PROGRAM MoveExtPos
VAR
	armState	:UINT:=0;
	chabustate	:UINT:=0;
	
	LeftArm_Right_ExtPosGen_Enable						:MC_ExtSetPointGenEnable;
	LeftArm_Right_ExtPosGen_Disable                     :MC_ExtSetPointGenDisable;
	LeftArm_Left_ExtPosGen_Enable                       :MC_ExtSetPointGenEnable;
	LeftArm_Left_ExtPosGen_Disable	                    :MC_ExtSetPointGenDisable;
	LeftArm_Wrist_ExtPosGen_Enable                      :MC_ExtSetPointGenEnable;
	LeftArm_Wrist_ExtPosGen_Disable	                    :MC_ExtSetPointGenDisable;
	
	RightArm_Right_ExtPosGen_Enable						:MC_ExtSetPointGenEnable;
	RightArm_Right_ExtPosGen_Disable                     :MC_ExtSetPointGenDisable;
	RightArm_Left_ExtPosGen_Enable                       :MC_ExtSetPointGenEnable;
	RightArm_Left_ExtPosGen_Disable	                    :MC_ExtSetPointGenDisable;
	RightArm_Wrist_ExtPosGen_Enable                      :MC_ExtSetPointGenEnable;
	RightArm_Wrist_ExtPosGen_Disable	                    :MC_ExtSetPointGenDisable;
	
	currentPosition_LeftArm				:Points;
	currentPosition_RightArm				:Points;

	//leftpoints						:ARRAY[0..5,0..1] OF LREAL:=[[-80,390],[390,880],[-80,390],[-80,880],[-80,390],[-400,830]];
	//rightpoints						:ARRAY[0..5,0..1] OF LREAL:=[[-80,390],[390,880],[-80,390],[-80,880],[-80,390],[-400,830]];	
	LeftArmWristTargetPos				:REAL;
	RightArmWristTargetPos				:REAL;	
	
	t			:LREAL:=0;
	delta_t		:LREAL:=0.0005;
	lx:LREAL;
	ly:LREAL;
	rx:LREAL;
	ry:LREAL;
	
	LeftArmAngle			:Angles;
	RightArmAngle			:Angles;


	
	

END_VAR

axis_LeftArm_Left();
axis_LeftArm_Right();
axis_LeftArm_Wrist();
axis_RightArm_Left();
axis_RightArm_Right();
axis_RightArm_Wrist();
ACT_ExtGen();


// 外部位置发生器失能
LeftArm_Right_ExtPosGen_Enable.Execute 		:= FALSE;
LeftArm_Right_ExtPosGen_Disable.Execute 	:= FALSE;
LeftArm_Left_ExtPosGen_Enable.Execute 		:= FALSE;
LeftArm_Left_ExtPosGen_Disable.Execute 		:= FALSE;
LeftArm_Wrist_ExtPosGen_Enable.Execute 		:= FALSE;
LeftArm_Wrist_ExtPosGen_Disable.Execute 	:= FALSE;	

RightArm_Right_ExtPosGen_Enable.Execute 	:= FALSE;
RightArm_Right_ExtPosGen_Disable.Execute 	:= FALSE;
RightArm_Left_ExtPosGen_Enable.Execute 		:= FALSE;
RightArm_Left_ExtPosGen_Disable.Execute 	:= FALSE;
RightArm_Wrist_ExtPosGen_Enable.Execute 	:= FALSE;
RightArm_Wrist_ExtPosGen_Disable.Execute 	:= FALSE;	


IF bAutoMovePosSet THEN

	
	CASE armState OF
		
		0:// 运动学正解出当前腕关节点坐标
			currentPosition_LeftArm 	:= LeftArmFK(axis_LeftArm_Right.NcToPlc.ActPos, axis_LeftArm_Left.NcToPlc.ActPos);
			currentPosition_RightArm 	:= RightArmFK(axis_RightArm_Right.NcToPlc.ActPos, axis_RightArm_Left.NcToPlc.ActPos);
			LeftArmWristTargetPos		:= LeftArmWristIK(axis_LeftArm_Right.NcToPlc.ActPos, axis_LeftArm_Left.NcToPlc.ActPos);
			RightArmWristTargetPos		:= RightArmWristIK(axis_RightArm_Right.NcToPlc.ActPos, axis_RightArm_Left.NcToPlc.ActPos);
			armState:=1;
		1:
			axis_LeftArm_Wrist_MoveAbs(
				Axis:= axis_LeftArm_Wrist, 
				Execute:= TRUE, 
				Position:= LeftArmWristTargetPos, 
				Velocity:= 0.5, 
				Acceleration:= 1, 
				Deceleration:= , 
				Jerk:= , 
				BufferMode:= , 
				Options:= , 
				Done=> , 
				Busy=> , 
				Active=> , 
				CommandAborted=> , 
				Error=> , 
				ErrorID=> );
			
			axis_RightArm_Wrist_MoveAbs(
				Axis:= axis_RightArm_Wrist, 
				Execute:= TRUE, 
				Position:= RightArmWristTargetPos, 
				Velocity:= 0.5, 
				Acceleration:= 1, 
				Deceleration:= , 
				Jerk:= , 
				BufferMode:= , 
				Options:= , 
				Done=> , 
				Busy=> , 
				Active=> , 
				CommandAborted=> , 
				Error=> , 
				ErrorID=> );
			IF axis_RightArm_Wrist_MoveAbs.Done = TRUE AND axis_LeftArm_Wrist_MoveAbs.Done = TRUE THEN
				armState:=2;
			END_IF

			
		2:
			LeftArm_Right_ExtPosGen_Enable.Execute 		:= TRUE;
			LeftArm_Left_ExtPosGen_Enable.Execute 		:= TRUE;
			LeftArm_Wrist_ExtPosGen_Enable.Execute 		:= TRUE;
			RightArm_Right_ExtPosGen_Enable.Execute 	:= TRUE;
			RightArm_Left_ExtPosGen_Enable.Execute 		:= TRUE;
			RightArm_Wrist_ExtPosGen_Enable.Execute 	:= TRUE;
			
			IF axis_LeftArm_Right.Status.ExtSetPointGenEnabled AND axis_LeftArm_Left.Status.ExtSetPointGenEnabled AND axis_RightArm_Right.Status.ExtSetPointGenEnabled AND axis_RightArm_Left.Status.ExtSetPointGenEnabled AND axis_LeftArm_Wrist.Status.ExtSetPointGenEnabled  AND axis_RightArm_Wrist.Status.ExtSetPointGenEnabled THEN

				CASE  chabustate OF
					0:
						lx	:=currentPosition_LeftArm.x+t*(-80-currentPosition_LeftArm.x);
						ly 	:=currentPosition_LeftArm.y+t*(390-currentPosition_LeftArm.y);
						rx	:=currentPosition_RightArm.x+t*(120-currentPosition_RightArm.x);
						ry 	:=currentPosition_RightArm.y+t*(370-currentPosition_RightArm.y);
						t	:= t+delta_t;
						IF t>=1 THEN
							LeftArm_Right_ExtPosGen_Enable.Execute := FALSE;
							LeftArm_Left_ExtPosGen_Enable.Execute := FALSE;
							RightArm_Right_ExtPosGen_Enable.Execute := FALSE;
							RightArm_Left_ExtPosGen_Enable.Execute := FALSE;
							chabustate:=1;
							t	:=0;
						END_IF

					1:

						lx	:=t*470-80;
						ly	:=390+t*490;
						rx	:=120+250*t;
						ry	:=370+510*t;
						t	:= t+delta_t;
						IF t >=1 THEN
							LeftArm_Right_ExtPosGen_Enable.Execute := FALSE;
							LeftArm_Left_ExtPosGen_Enable.Execute := FALSE;
							RightArm_Right_ExtPosGen_Enable.Execute := FALSE;
							RightArm_Left_ExtPosGen_Enable.Execute := FALSE;
							chabustate := 2;
							t:=0;
						END_IF
					2:
						lx	:=390-t*470;
						ly	:=880-t*490;
						rx	:=370-250*t;
						ry	:=880-510*t;
						t	:= t+delta_t;
						IF t>=1 THEN
							LeftArm_Right_ExtPosGen_Enable.Execute := FALSE;
							LeftArm_Left_ExtPosGen_Enable.Execute := FALSE;
							RightArm_Right_ExtPosGen_Enable.Execute := FALSE;
							RightArm_Left_ExtPosGen_Enable.Execute := FALSE;
							chabustate := 3;
							t:=0;
						END_IF
					3:
						lx := -80;
						ly := 390+490*t;
						rx := 120;
						ry := 370+510*t;
						t:=t+delta_t;
						IF t>= 1 THEN
							LeftArm_Right_ExtPosGen_Enable.Execute := FALSE;
							LeftArm_Left_ExtPosGen_Enable.Execute := FALSE;
							RightArm_Right_ExtPosGen_Enable.Execute := FALSE;
							RightArm_Left_ExtPosGen_Enable.Execute := FALSE;
							chabustate	:=4;
							t:=0;
						END_IF
					4:
						lx := -80;
						ly := 880-490*t;
						rx := 120;
						ry := 880-510*t;
						t:= t+delta_t;
						IF t>=1 THEN
							LeftArm_Right_ExtPosGen_Enable.Execute := FALSE;
							LeftArm_Left_ExtPosGen_Enable.Execute := FALSE;
							RightArm_Right_ExtPosGen_Enable.Execute := FALSE;
							RightArm_Left_ExtPosGen_Enable.Execute := FALSE;
							chabustate := 5;
							t:=0;
						END_IF
					5:
						lx := -80-320*t;
						ly := 390+440*t;
						rx := 120-450*t;
						ry := 370+480*t;
						t:=t+delta_t;
						IF t>= 1 THEN
							LeftArm_Right_ExtPosGen_Enable.Execute := FALSE;
							LeftArm_Left_ExtPosGen_Enable.Execute := FALSE;
							RightArm_Right_ExtPosGen_Enable.Execute := FALSE;
							RightArm_Left_ExtPosGen_Enable.Execute := FALSE;
							chabustate	:=6;
							t:=0;
						END_IF
					6:
						lx := -400+320*t;
						ly := 830-440*t;
						rx := -330+450*t;
						ry := 850-480*t;
						t:= t+delta_t;
						IF t>=1 THEN
							LeftArm_Right_ExtPosGen_Enable.Execute := FALSE;
							LeftArm_Left_ExtPosGen_Enable.Execute := FALSE;
							RightArm_Right_ExtPosGen_Enable.Execute := FALSE;
							RightArm_Left_ExtPosGen_Enable.Execute := FALSE;
							chabustate := 1;
							t:=0;
						END_IF

				END_CASE
				
				LeftArmAngle := LeftArmIK(lx,ly);
				LeftArmWristTargetPos := LeftArmWristIK(LeftArmAngle.theta1_right, LeftArmAngle.theta2_left);
				
				RightArmAngle := RightArmIK(rx,ry);
				RightArmWristTargetPos := RightArmWristIK(RightArmAngle.theta1_right, RightArmAngle.theta2_left);
					
	
				
				LeftArm_Right_ExtPosGen_Enable.Execute := TRUE;
				LeftArm_Left_ExtPosGen_Enable.Execute := TRUE;
				RightArm_Right_ExtPosGen_Enable.Execute := TRUE;
				RightArm_Left_ExtPosGen_Enable.Execute := TRUE;
				
				MC_ExtSetPointGenFeed(
					Position:= LeftArmAngle.theta1_right, 
					Velocity:= 0.005,  
					Acceleration:= 0.01,  
					Direction:= 1, 
					Axis:= axis_LeftArm_Right);
		
				MC_ExtSetPointGenFeed(
					Position:= LeftArmAngle.theta2_left, 
					Velocity:= 0.005,  
					Acceleration:= 0.001,  
					Direction:= 1, 
					Axis:= axis_LeftArm_Left);
				
				MC_ExtSetPointGenFeed(
					Position:= RightArmAngle.theta1_right, 
					Velocity:= 0.005,  
					Acceleration:= 0.01,  
					Direction:= 1, 
					Axis:= axis_RightArm_Right);
		
				MC_ExtSetPointGenFeed(
					Position:= RightArmAngle.theta2_left, 
					Velocity:= 0.005,  
					Acceleration:= 0.001,  
					Direction:= 1, 
					Axis:= axis_RightArm_left);
												
				MC_ExtSetPointGenFeed(
					Position:= LeftArmWristTargetPos, 
					Velocity:= 0.5, 
					Acceleration:= 1, 
					Direction:= 1, 
					Axis:= axis_LeftArm_Wrist);

					
				MC_ExtSetPointGenFeed(
					Position:= RightArmWristTargetPos, 
					Velocity:= 5, 
					Acceleration:= 10, 
					Direction:= 1, 
					Axis:= axis_RightArm_Wrist);
				

			END_IF
	
	END_CASE




END_IF

ACTION ACT_ExtGen:
LeftArm_Right_ExtPosGen_Enable(
	Axis:= axis_LeftArm_Right, 
	Execute:= LeftArm_Right_ExtPosGen_Enable.Execute, 
	Position:= , 
	PositionType:= , 
	Done=> , 
	Busy=> , 
	Error=> , 
	ErrorID=> , 
	Enabled=> );
	
LeftArm_Right_ExtPosGen_Disable(
	Axis:= axis_LeftArm_Right, 
	Execute:= LeftArm_Right_ExtPosGen_Disable.Execute, 
	Done=> , 
	Busy=> , 
	Error=> , 
	ErrorID=> , 
	Enabled=> );
	
LeftArm_Left_ExtPosGen_Enable(
	Axis:= axis_LeftArm_Left, 
	Execute:= LeftArm_Left_ExtPosGen_Enable.Execute, 
	Position:= , 
	PositionType:= , 
	Done=> , 
	Busy=> , 
	Error=> , 
	ErrorID=> , 
	Enabled=> );
	
LeftArm_Left_ExtPosGen_Disable(
	Axis:= axis_LeftArm_Left, 
	Execute:= LeftArm_Left_ExtPosGen_Disable.Execute, 
	Done=> , 
	Busy=> , 
	Error=> , 
	ErrorID=> , 
	Enabled=> );
	
LeftArm_Wrist_ExtPosGen_Enable(
	Axis:= axis_LeftArm_Wrist, 
	Execute:= LeftArm_Wrist_ExtPosGen_Enable.Execute, 
	Position:= , 
	PositionType:= , 
	Done=> , 
	Busy=> , 
	Error=> , 
	ErrorID=> , 
	Enabled=> );
	
LeftArm_Wrist_ExtPosGen_Disable(
	Axis:= axis_LeftArm_Wrist, 
	Execute:= LeftArm_Wrist_ExtPosGen_Disable.Execute, 
	Done=> , 
	Busy=> , 
	Error=> , 
	ErrorID=> , 
	Enabled=> );
	
RightArm_Right_ExtPosGen_Enable(
	Axis:= axis_RightArm_Right, 
	Execute:= RightArm_Right_ExtPosGen_Enable.Execute, 
	Position:= , 
	PositionType:= , 
	Done=> , 
	Busy=> , 
	Error=> , 
	ErrorID=> , 
	Enabled=> );
	
RightArm_Right_ExtPosGen_Disable(
	Axis:= axis_RightArm_Right, 
	Execute:= RightArm_Right_ExtPosGen_Disable.Execute, 
	Done=> , 
	Busy=> , 
	Error=> , 
	ErrorID=> , 
	Enabled=> );
	
RightArm_Left_ExtPosGen_Enable(
	Axis:= axis_RightArm_Left, 
	Execute:= RightArm_Left_ExtPosGen_Enable.Execute, 
	Position:= , 
	PositionType:= , 
	Done=> , 
	Busy=> , 
	Error=> , 
	ErrorID=> , 
	Enabled=> );
	
RightArm_Left_ExtPosGen_Disable(
	Axis:= axis_RightArm_Left, 
	Execute:= RightArm_Left_ExtPosGen_Disable.Execute, 
	Done=> , 
	Busy=> , 
	Error=> , 
	ErrorID=> , 
	Enabled=> );
	
RightArm_Wrist_ExtPosGen_Enable(
	Axis:= axis_RightArm_Wrist, 
	Execute:= RightArm_Wrist_ExtPosGen_Enable.Execute, 
	Position:= , 
	PositionType:= , 
	Done=> , 
	Busy=> , 
	Error=> , 
	ErrorID=> , 
	Enabled=> );
	
RightArm_Wrist_ExtPosGen_Disable(
	Axis:= axis_RightArm_Wrist, 
	Execute:= RightArm_Wrist_ExtPosGen_Disable.Execute, 
	Done=> , 
	Busy=> , 
	Error=> , 
	ErrorID=> , 
	Enabled=> );
END_ACTION

END_PROGRAM

(* stored: Version 1.1.0.1, ProductVersion 3.1.4024.14
   POU MoveExtPos: Id {14b2fa12-99b5-447e-ad50-13da07e623f6}, SpecialFunc None
   Action ACT_ExtGen: Id {497ad5f0-c9f3-4530-aa78-af8a1b8cb86f} *)
